// TIA Portal V15.1 export
// export: Created 2022-12-20T09:13:23.260207Z, ExportSetting None, DisplayName Totally Integrated Automation Portal, DisplayVersion V15.1 Update 1, DisplayName TIA Portal Openness, DisplayVersion V15.1, DisplayName SINAMICS Startdrive Advanced, DisplayVersion V15.1, DisplayName G130, G150, S120, S150, SINAMICS MV, S210, DisplayVersion V15.1, DisplayName G110M, G120, G120C, G120D, G120P, DisplayVersion V15.1, DisplayName STEP 7 Professional, DisplayVersion V15.1 Update 1, DisplayName STEP 7 Safety, DisplayVersion V15.1, DisplayName WinCC Professional, DisplayVersion V15.1 Update 1, DisplayName SIMATIC Visualization Architect, DisplayVersion V15.1
FUNCTION_BLOCK "SA01_DAQ_FB"   // FB903, FBD
TITLE = SA01_DAQ_FB
{ S7_Optimized_Access := 'FALSE' }
// The block is used to control the data acquisition such as part counters, cycle time counters
// stored: AutoNumber false, SetENOAutomatically False
   VAR
      "SA01-PC01" : "CM_Counter_FB";   // Counter SA01
      "xxx-xxxxx-CT01" : "CM_Cycle_Timer_FB";   // Cycle Time xxxxx
      "SA01-CT01" : "CM_Cycle_Timer_FB";   // Cycle Time SA01
   END_VAR
BEGIN

REGION Network 1: *** Cycle Time ***
END_REGION

REGION Network 2: ******* Stxx *******
END_REGION

REGION Network 3: Cycle Time xxxx
   // Cycle Time 10FX01
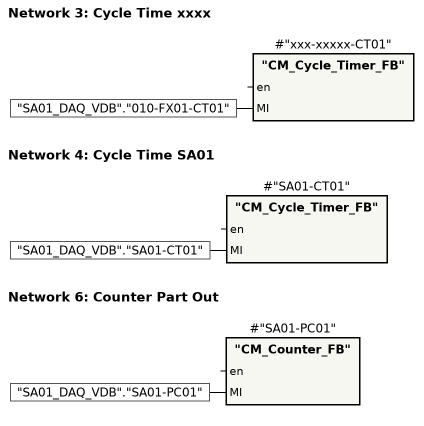
   #"xxx-xxxxx-CT01"(MI := "SA01_DAQ_VDB"."010-FX01-CT01");   // "CM_Cycle_Timer_FB"
END_REGION

REGION Network 4: Cycle Time SA01
   // Cycle Time SA01
   #"SA01-CT01"(MI := "SA01_DAQ_VDB"."SA01-CT01");   // "CM_Cycle_Timer_FB"
END_REGION

REGION Network 5: *** Counter ***
END_REGION

REGION Network 6: Counter Part Out
   // Counter Part Out
   #"SA01-PC01"(MI := "SA01_DAQ_VDB"."SA01-PC01");   // "CM_Counter_FB"
END_REGION
END_FUNCTION_BLOCK
